// Mitsubishi GX Works2 project: Start_5_Lan_Du_5_Phoi_Vs_Timer   PLC: FX2N/FX2NC

PROGRAM MAIN
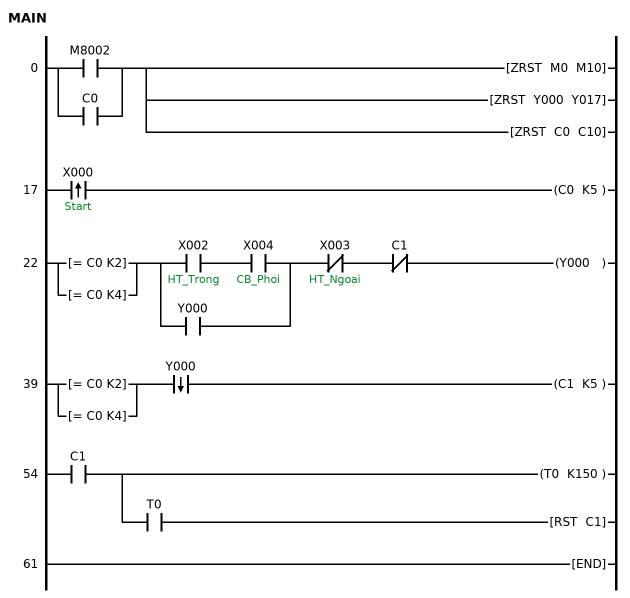
0     LD      M8002
      OR      C0
      ZRST    M0 M10
      ZRST    Y000 Y017
      ZRST    C0 C10
17    LDP     X000  ; Start
      OUT     C0 K5
22    LD=     C0 K2
      OR=     C0 K4
      LD      X002  ; HT_Trong
      AND     X004  ; CB_Phoi
      OR      Y000
      ANB
      ANI     X003  ; HT_Ngoai
      ANI     C1
      OUT     Y000
39    LD=     C0 K2
      OR=     C0 K4
      ANDF    Y000
      OUT     C1 K5
54    LD      C1
      OUT     T0 K150
      AND     T0
      RST     C1
61    END
END_PROGRAM

// device comments not shown above
X001  ; Reset
